(* IEC 61131-3 sources: AdvIecChk/AdvIecChk/AdvIecChk/V1.00.0, 2 files *)

(* ---- AdvIecChk.fun ---- *)
(********************************************************************
 * COPYRIGHT --
 ********************************************************************
 * Library: IecCheck
 * File: IecCheck.fun
 * Author: adamsm
 * Created: October 03, 2012
 ********************************************************************
 * Functions and function blocks of library IecCheck
 ********************************************************************)

FUNCTION CheckDivDWord : UDINT (* Check divisor for DINT and UDINT division *)
	VAR_INPUT
		divisor : UDINT;
	END_VAR
END_FUNCTION

FUNCTION CheckDivWord : UINT (* Check divisor for INT and UINT division *)
	VAR_INPUT
		divisor : UINT;
	END_VAR
END_FUNCTION

FUNCTION CheckDivByte : USINT (* Check divisor for SINT and USINT division *)
	VAR_INPUT
		divisor : USINT;
	END_VAR
END_FUNCTION

FUNCTION CheckDivReal : REAL (* Check divisor for REAL division *)
	VAR_INPUT
		divisor : REAL;
	END_VAR
END_FUNCTION

FUNCTION CheckDivLReal : LREAL (* Check divisor for LREAL division, not available for SG3 and SGC *)
	VAR_INPUT
		divisor : LREAL;
	END_VAR
END_FUNCTION

FUNCTION CheckBounds : DINT (* Check range for array access *)
	VAR_INPUT
		index : DINT;
		lower : DINT;
		upper : DINT;
	END_VAR
	VAR
		LowString : STRING[4];
		UpString : STRING[4];
		IndexString : STRING[4];
		text : STRING[80];
	END_VAR
END_FUNCTION

FUNCTION CheckRange : DINT (* Check range for enumeration *)
	VAR_INPUT
		value : DINT;
		lower : DINT;
		upper : DINT;
	END_VAR
END_FUNCTION

FUNCTION CheckSignedSubrange : DINT (* Check range for subrange of signed data types *)
	VAR_INPUT
		value : DINT;
		lower : DINT;
		upper : DINT;
	END_VAR
END_FUNCTION

FUNCTION CheckUnsignedSubrange : UDINT (* Check range for subrange of unsigned data types *)
	VAR_INPUT
		value : UDINT;
		lower : UDINT;
		upper : UDINT;
	END_VAR
END_FUNCTION

FUNCTION CheckReadAccess : UDINT (* Check address when reading dynamic variables *)
	VAR_INPUT
		address : UDINT;
	END_VAR
END_FUNCTION

FUNCTION CheckWriteAccess : UDINT (* Check address when writing dynamic variables *)
	VAR_INPUT
		address : UDINT;
	END_VAR
END_FUNCTION

FUNCTION MakeEntry : UDINT (* Makes an entry (log book entry) in the error log book *)
	VAR_INPUT
		number : UINT;
		index : DINT;
		text : STRING[50];
	END_VAR
	VAR
		taskname : STRING[30];
		group : USINT;
		status_name : UINT;
		out_text : STRING[80];
		pv_adr : UDINT;
		data_len : UDINT;
		SectionString : STRING[80];
		SectionData : DINT;
	END_VAR
END_FUNCTION

(* ---- AdvIecChk.st ---- *)
(********************************************************************
 * COPYRIGHT --
 ********************************************************************
 * Library: IecCheck
 * Author: adamsm
 * Created: August 20, 2012
 ********************************************************************
 * Implementation of library IecCheck
 ********************************************************************)

(* Check divisor for DINT and UDINT division *)
FUNCTION CheckDivDWord
	IF divisor=0 THEN
		CheckDivDWord:=1;
		MakeEntry(55555,divisor,'Divide by Zero - Double Word');
	ELSE
		CheckDivDWord:=divisor;
	END_IF
END_FUNCTION

(* Check divisor for INT and UINT division *)
FUNCTION CheckDivWord
	IF divisor=0 THEN
		CheckDivWord:=1;
		MakeEntry(55555,divisor,'Divide by Zero - Word');
	ELSE
		CheckDivWord:=divisor;
	END_IF
END_FUNCTION

(* Check divisor for SINT and USINT division *)
FUNCTION CheckDivByte
	IF divisor=0 THEN
		CheckDivByte:=1;
		MakeEntry(55555,divisor,'Divide by Zero - Byte');
	ELSE
		CheckDivByte:=divisor;
	END_IF
END_FUNCTION

(* Check divisor for REAL division *)
FUNCTION CheckDivReal
	IF divisor=0 THEN
		CheckDivReal:=1;
		MakeEntry(55555,0,'Divide by Zero - Real');
	ELSE
		CheckDivReal:=divisor;
	END_IF
END_FUNCTION

(* Check divisor for LREAL division *)
FUNCTION CheckDivLReal
	IF divisor=0 THEN
		CheckDivLReal:=1;
		MakeEntry(55555,0,'Divide by Zero - Long Real');
	ELSE
		CheckDivLReal:=divisor;
	END_IF
END_FUNCTION

(* Check range for enumeration *)
FUNCTION CheckRange
	IF value < lower THEN
		CheckRange := lower;
		MakeEntry(55555,value,'ENUM-Check Low');
	ELSIF value > upper THEN
		CheckRange := upper;
		MakeEntry(55555,value,'ENUM-Check High');
	ELSE
		CheckRange := value;
	END_IF
END_FUNCTION

(* Check range for subrange of signed data types *)
FUNCTION CheckSignedSubrange
	IF value < lower THEN
		CheckSignedSubrange := lower;
		MakeEntry(55555,value,'CheckSignedSubrange Low');
	ELSIF value > upper THEN
		CheckSignedSubrange := upper;
		MakeEntry(55555,value,'CheckSignedSubrange High');
	ELSE
		CheckSignedSubrange := value;
	END_IF
END_FUNCTION

(* Check range for subrange of unsigned data types *)
FUNCTION CheckUnsignedSubrange
	IF value < lower THEN
		CheckUnsignedSubrange := lower;
		MakeEntry(55555,value,'CheckUnsignedSubrange Low');
	ELSIF value > upper THEN
		CheckUnsignedSubrange := upper;
		MakeEntry(55555,value,'CheckUnsignedSubrange High');
	ELSE
		CheckUnsignedSubrange := value;
	END_IF
END_FUNCTION

(* Check address when reading dynamic variables *)
FUNCTION CheckReadAccess
	IF address=0 THEN
		(* TODO: Insert an appropriate code, see AutomationStudio help for further information *)
		MakeEntry(55555,address,'Attempt to read from address of zero / NULL');
	END_IF

	CheckReadAccess:=0;
END_FUNCTION

(* Check address when writing dynamic variables *)
FUNCTION CheckWriteAccess
	IF address=0 THEN
		(* TODO: Insert an appropriate code, see AutomationStudio help for further information *)
		MakeEntry(55555,address,'Attempt to write to address of zero / NULL');
	END_IF

	CheckWriteAccess:=0;
END_FUNCTION

FUNCTION CheckBounds (* Check range for array access *)
	IF index < lower OR index > upper THEN
		itoa(lower, ADR(LowString));
		itoa(upper, ADR(UpString));
		itoa(index, ADR(IndexString));
		CheckBounds := upper;
		strcpy(ADR(text),ADR('Array Index '));
		strcat(ADR(text),ADR(IndexString));
		strcat(ADR(text),ADR(' is outside ['));
		strcat(ADR(text),ADR(LowString));
		strcat(ADR(text),ADR('..'));
		strcat(ADR(text),ADR(UpString));
		strcat(ADR(text),ADR(']'));
		MakeEntry(55555,index,text);
	ELSE
		CheckBounds := index;
	END_IF
END_FUNCTION

FUNCTION MakeEntry (* Makes a log book entry *)
	status_name := ST_name(0,ADR(taskname),ADR(group));
	PV_xgetadr(ADR('gIecChkSec'), ADR(pv_adr), ADR(data_len));
	IF pv_adr > 0 AND data_len > 0 THEN
		memcpy(ADR(SectionData),pv_adr,data_len);
		itoa(SectionData,ADR(SectionString));
	END_IF

	strcpy(ADR(out_text),ADR(text));
	strcat(ADR(out_text),ADR(' in task "'));
	strcat(ADR(out_text),ADR(taskname));
	strcat(ADR(out_text),ADR('" Section:'));
	strcat(ADR(out_text),ADR(SectionString));
	MakeEntry := ADR(out_text);
	ERRxfatal(number,index,ADR(out_text));
END_FUNCTION
